Fanuc KAREL source: kf00044.KL

PROGRAM KF00044
%STACKSIZE=65535
%PRIORITY=65535
%NOLOCKGROUP
TYPE
REC_T=STRUCTURE
VALUE : INTEGER
FLAG : BOOLEAN
ENDSTRUCTURE
VAR
I : INTEGER
J : INTEGER
X : REAL
Y : REAL
B : BOOLEAN
C : BOOLEAN
TXT : STRING[80]
TXT2 : STRING[80]
AI : ARRAY[4] OF INTEGER
BI : ARRAY[4] OF INTEGER
P : XYZWPR
JP : JOINTPOS9
PF : POSITION
V1 : VECTOR
V2 : VECTOR
STATUS : INTEGER
REC : REC_T
REC2 : REC_T
BEGIN
REC.VALUE=7
-- UNRESOLVED_PC line 29 opcodes [22 22 30] marker_code=20
END KF00044
